// TIA Portal V17 export
// export: Created 2024-06-14T09:52:48.268429Z, ExportSetting WithDefaults, DisplayName Totally Integrated Automation Portal, DisplayVersion V17, DisplayName TIA Portal Openness, DisplayVersion V17, DisplayName TIA Portal Version Control Interface, DisplayVersion V17, DisplayName Simotion SCOUT TIA, DisplayVersion 5.4.3.0, DisplayName SINAMICS Startdrive Advanced, DisplayVersion V17 SP1 Update 1, DisplayName SINAMICS Startdrive G110M, G120, G120C, G120D, G120P, G115D, DisplayVersion V17 SP1 Update 1, DisplayName SINAMICS Startdrive G130, G150, S120, S150, SINAMICS MV, S210, DisplayVersion V17 SP1 Update 1, DisplayName STEP 7 Professional, DisplayVersion V17, DisplayName STEP 7 Safety, DisplayVersion V17, DisplayName WinCC Professional, DisplayVersion V17
DATA_BLOCK "FILLING_STATION4_DB"   // DB500
VERSION : 0.1
// stored: AutoNumber false, DBAccessibleFromOPCUA true, InstanceOfName FILLING_STATION4_FB, InstanceOfType FB
"FILLING_STATION4_FB"
   // VAR
   //    STATION4_S1 { S7_SetPoint := 'True'} : "LPG_FILLING_FB";
   //    STATION4_S2 { S7_SetPoint := 'True'} : "LPG_FILLING_FB";
   //    STATION4_S3 { S7_SetPoint := 'True'} : "LPG_FILLING_FB";
   //    STATION4_S4 { S7_SetPoint := 'True'} : "LPG_FILLING_FB";
   //    STATION4_S5 { S7_SetPoint := 'True'} : "LPG_FILLING_FB";
   //    STATION4_S6 { S7_SetPoint := 'True'} : "LPG_FILLING_FB";
   //    FILLING_STATION4 { S7_SetPoint := 'True'} : "FILLING_FB";
   //    FILL_SEQ_STARTED { S7_SetPoint := 'True'} : Array[1..6] of Bool;
   //    FILLING_DONE : Array[1..6] of Bool;
   // END_VAR
BEGIN
END_DATA_BLOCK
